{attribute addProperty BoxType "EL3692-0000-0017"}
{attribute addProperty Id "ValueAT %I*REAL324"}
{attribute addProperty CRC "1594033361"}
{attribute addProperty SizeInBites "32"}
{attribute addProperty SizeInBytes "4"}
TYPE SAI_Inputs_Real_Channel_5F0304D1 :
STRUCT
	{attribute addProperty Name "Value"}
	Value AT %I* : REAL;
END_STRUCT
END_TYPE

(* stored: Version 1.2.0.0, ProductVersion 3.1.4024.9
   DUT SAI_Inputs_Real_Channel_5F0304D1: Id {0f92adb0-be45-4ae7-a51f-287d2a862352} *)
